PROGRAM TCPCom
VAR
END_VAR

PRG_TCPIP();

END_PROGRAM

(* stored: Version 1.1.0.1, ProductVersion 3.1.4024.12
   POU TCPCom: Id {fb9fad86-a609-4e23-8150-11d22b07403a}, SpecialFunc None *)
